(* CODESYS project lclsvacuum.library
   Company: SLAC
   Title: LCLSVacuumLib
   Description: No serial drivers exist in this library. Need LCLSVacuumSerialDrivers for that.
      1.2.0 ecat diagnostic
      1.2.1 added the ecat lib in here
      1.2.2 adding the ratio check function for valve interlocking
      1.3.6 added 275 & 500 gauges, minor changes
      1.4.0 added a normally open gate valve structure and FB
      1.5.0 added error and warning codes to ptm structure for pfeiffers
      1.5.1 seamless override open/close on vgc during transition from override to normal mode.
      1.7.0 ST_PTM now uses inheritence model.  Started implementing Ebara support.
      1.8.0 Moved to seperate functions for 937A and 937B controllers.
   Placeholder: LCLSVacuumLib
   Author: Alex Wallace & Scott Stubbs
   Version: 1.10.3

Project tree, tasks and I/O mapping:
  libraries: Tc2_EtherCAT, * (Beckhoff Automation GmbH); Tc2_Standard, * (Beckhoff Automation GmbH); Tc2_System, * (Beckhoff Automation GmbH); Tc2_TcpIp, * (Beckhoff Automation GmbH); Tc2_Utilities, * (Beckhoff Automation GmbH); Tc3_Interfaces, * (Beckhoff Automation GmbH); Tc3_Module, * (Beckhoff Automation GmbH)
  Data types/
    Gauges/
      data type E_PressureState
      data type Gauge_Type
      data type ST_VG
    Logger/
      data type E_MesgSevr
      data type E_MessengerState
      data type E_Subsystem
    Misc/
      data type ST_fbDiagnostics
      data type System_Struct
    Pumps/
      data type ST_AgilentControlStatus
      data type ST_EbaraDryPump
      data type ST_EbaraPTM
      data type ST_LeyboldPTM
      data type ST_PfeifferPTM
      data type ST_PTM
      data type ST_RoughPump
    Valves/
      data type E_VCN
      data type E_VGC
      data type ST_VCC
      data type ST_VCN
      data type ST_VGC
      data type ST_VGC_NO
      data type ST_VRC
    data type ISG_Struct
    data type ST_Encoder
    data type ST_LaserGate
    data type UpStrInVac_Struct
    data type UpStrOutVac_Struct
  Global Variables/
    global variables Constants
    global variables Global_Variables
    global variables GVL_Logger
  POUs/
    Functions/
      Gauge FB/
        function block FB_275 [ST]
        function block FB_500 [ST]
        function block FB_903 [ST]
        function block FB_907 [ST]
        function block FB_909 [ST]
        function block FB_925 [ST]
        function block FB_937A_VG [ST]
        function block FB_937B_VG [ST]
        function block FB_972 [ST]
        function block FB_Dumb_Gauge [ST]
        function block FB_GCM [ST]
        function block FB_GGO [ST]
        function block FB_GGO_dep [ST]
        function block FB_PressureState [ST]
      Pumps/
        function block FB_EbaraDryPump [ST]
        function block FB_PTM_Agilent [ST]
        function block FB_PTM_Ebara [ST]
        function block FB_PTM_LeyboldTD20Classic [ST]
        function block FB_PTM_MagDriveDigital [ST]
        function block FB_PTM_Pfeiffer [ST]
      Valve FB/
        function F_TURBO_VRC_ILK [ST]
        function F_VALVE_REL_ILK [ST]
        function F_VRC_DIODE_ILK [ST]
        function block FB_VCC [ST]
        function block FB_VCN [ST]
        function block FB_VGC [ST]: ACT_ResetAlarms
        function block FB_VGC_NO [ST]: ACT_ResetAlarms
        function block FB_VRC [ST]
        function block FB_VRC_OK_CLS [ST]
      function block FB_EcatDiag [ST]
      function block FB_Index [ST]: Dec, Inc, ValInc
    Logger/
      function block FB_Logger [ST]: Manager, SocketSendTo
      function block FB_LogMessage [ST]
      function SYSTEM_TIME_TO_RFC3339 [ST]
    program LOGGER [ST]
    program MAIN [ST]
  Version/
    global variables Global_Version
  Visualizations/
  00000000-0000-0000-0000-000000000000|LCLSVacuum.tmc
  LCLSVacuum.tmc
*)

// Data types/Gauges/E_PressureState
TYPE E_PressureState :
(
	Valid := gc_GaugeValidState,
	ValidHi	:= 1, //gc_GaugeValidState + 1,
	ValidLo	:= 2, //gc_GaugeValidState + 2,
	
	// Invalid states
	Invalid	:= -1, //gc_GaugeValidState - 1,
	Disconnected	:=	-2, //gc_GaugeValidState -2,
	OoR	:= -6, //gc_GaugeValidState -6,
	// Ion gauges
	Off		:= -3, //gc_GaugeValidState - 3,
	Starting	:= -4 //gc_GaugeValidState - 4
) INT;
END_TYPE

// Data types/Gauges/Gauge_Type
TYPE Gauge_Type: ( 
PG722B := 0, 
IG903 := 1 , 
PG907 := 2 , 
IG909:= 3 ,
PG925 := 4 );
(* This enumeration should match up with the EDM MUX button on the vacuum gauge expert controls screen *)
END_TYPE

// Data types/Gauges/ST_VG
TYPE ST_VG :
STRUCT
	/// A general gauge structure is used to make the rest of the interlocking simpler. There are some parameters for cold cathodes that are not used by pirani.
	///These features aren't disabled, they just aren't used, think child/parent classes. 
	/// Readbacks 
	rPRESS: REAL; //This is the human-readable pressure
	iPRESS_R: INT;
	xAT_VAC: BOOL;
	xPRESS_OK: BOOL;
	wState	:	WORD; //current gauge state, to be used as replacement for press OK bit in the future.
	(* 00 controller not on
		01 normal, aka pressure OK
		02 LO, pressure too low
		03 HI, pressure too high
		04 Gauge disconnected, HV off, no sensor detected, controller powering up
		05 cold cathode warming up
		*)
	eState	:	E_PressureState;
	
	/// Controls 
	xHV_DIS: BOOL;
	xHV_SW: BOOL;
	wHV_RO: WORD;
	
	/// Bakeout bit 
	xBAKEOUT: BOOL;
	
	eTYPE: Gauge_Type := PG907;
	iTYPE : INT := 0;
	wPG: WORD;
	
	/// Turn on Timers for cold cathode warmup 
	xTurnOnTime: BOOL;
	/// At vacuum setpoint for all gauges
	rVAC_SP: REAL := 0.5;
	/// Protection setpoint for ion gauges at which the gauge turns off, not used for pirani 
	rPRO_SP: REAL := 0.01;
	/// Protection setpoint hysteresis 
	rHYS_PR: REAL;
	/// Full scale pressure in Torr for baratron pressure conversion 
	rFULL_SCALE: REAL := 1000;
END_STRUCT
END_TYPE

// Data types/Logger/E_MesgSevr
TYPE E_MesgSevr :
(
	Emergency := 0, //system is unusable
	Alert	:= 1,	//action must be taken immediately
	Critical:= 2,	//critical conditions
	Error	:= 3,	//error conditions
	Warning	:= 4,	//warning conditions
	Notice	:= 5,	//normal but significant condition
	Info	:= 6,	//informational messages
	Debug	:= 7	//debug-level messages
) WORD;
END_TYPE

// Data types/Logger/E_MessengerState
TYPE E_MessengerState :
(
	Init := 0,
	CreateSocket	:= 1,
	Active	:= 2,
	CloseSocket := 3,
	Err	:= 10
);
END_TYPE

// Data types/Logger/E_Subsystem
TYPE E_Subsystem :
(
	NILVALUE := 0,
	VACUUM := 1,
	MPS := 2,
	MOTION := 3,
	FIELDBUS := 4,
	SDS := 5
)WORD;
END_TYPE

// Data types/Misc/ST_fbDiagnostics
TYPE ST_fbDiagnostics :
STRUCT
	asResults	:	ARRAY [1..20] OF STRING;
	resultIdx	:	FB_Index := (
		InitVal := 1,
		UpperLimit := 20
	);
	fString	:	FB_FormatString;
END_STRUCT
END_TYPE

// Data types/Misc/System_Struct
TYPE System_Struct :
STRUCT

	xswAlmRst 		: BOOL;(* Global Alarm Reset - EPICS Command *)
	xAtVacuum 	    : BOOL;(* System At Vacuum *)
	xFirstScan	    : BOOL; (* Bit set for one scan only during startup. Used for initialization. *)
	xOverrideMode	: BOOL; //This bit is set when using the override features of the system
	xIOState        : BOOL; (* ECat Bus Health *)

END_STRUCT
END_TYPE

// Data types/Pumps/ST_AgilentControlStatus
TYPE ST_AgilentControlStatus :
STRUCT

(* Inputs *)
	xdiR1   		:  BOOL;
	xdiLSpd 		:  BOOL;
	xdiStart		:  BOOL;
	xdiR2   		:  BOOL;
	xdiFlt   	:  BOOL;
	xswStart		:  BOOL;
	xswLSpd 		:  BOOL;
	xswSS   		:  BOOL;
	xilkStart	:  BOOL;
	xilkLSpd   	:  BOOL;
	xilkEnb   	:  BOOL;
	xilkSS   	:  BOOL;
	xAlmRst   	:  BOOL;

(* Outputs *)
	xdoStart	:  BOOL;
	xdoLSpd	:  BOOL;
	xdoEnb	:  BOOL;
	xdoSS	:  BOOL;

(* Alarm Outputs *)
	xalmFlt		:  BOOL;
	xalmStart	:  BOOL;
	xalmLSpd		:  BOOL;
	xalmSS		:  BOOL;
	xAlmSum		: BOOL;


END_STRUCT
END_TYPE

// Data types/Pumps/ST_EbaraDryPump
TYPE ST_EbaraDryPump EXTENDS ST_RoughPump :
STRUCT
(* Extension of the rough pump archetype for ebara 
Applicable to: 
EV-S20
EV-S50
EV-S100
EV-S200
*)

//Controls
q_xMPStart	:	BOOL; //Main Pump start
q_xBPStart	:	BOOL; // Booster Pump start (this can be started by the pump automatically)

xBPIlk	:	BOOL;	//Booster pump interlock
rBPIlkSP	:	REAL := 30; //Booster pump pressure setpoint
tonBP	:	TON := (PT:=T#5S); //Timer for pressure and valve stability


//Readbacks
i_xMPStatus	:	BOOL; //MP status
i_xBPStatus	:	BOOL; //BP status
i_xWarning	:	BOOL; //Warning status
i_xAlarm	:	BOOL; //Alarm, maps to error
i_xRemote	:	BOOL; //Remote control status


END_STRUCT
END_TYPE

// Data types/Pumps/ST_EbaraPTM
TYPE ST_EbaraPTM EXTENDS ST_PTM :
STRUCT
(* Extension of the PTM archetype for Ebara turbo controllers 
Applicable to: 
ETC series
*)
//Controls
i_xStart   : BOOL; //Momentary start switch
i_xStop    : BOOL; //Momentary stop switch
//i_xReset   : BOOL; //Momentary reset switch - resets protection functions
q_xStart   : BOOL; //Outputs - FB decides if these are actually set
q_xStop    : BOOL;
q_xReset   : BOOL;
q_xProtection : BOOL; //NC. If opened, pump will decelerate/not start

iq_xSpeedSet    : BOOL; //Request to set speed
q_iSpeedSet   : DINT; //Requested speed (min. 100 RPM)

i_xOverride   : BOOL; //Override mode - ignores interlocks

//Readbacks - also has Accel/At speed/Decel/Fault/Cur Speed (min 100RPM)
i_xRotate : BOOL; //If open, pump is rotating
i_xDecel  : BOOL; //If closed, brake engaged (pump decelerating)
i_xNCFault  : BOOL; //Normally closed fault wiring. If false, there is a fault, or cable is unplugged.
i_iRawSpeed	:	INT; //Raw pump speed from analog input

END_STRUCT
END_TYPE

// Data types/Pumps/ST_LeyboldPTM
TYPE ST_LeyboldPTM EXTENDS ST_PTM :
STRUCT
(* Extension of the PTM archetype for Oerlikon turbo controllers 
Applicable to: 
Mag Drive Digital
Mag Drive S
More?
*)
//Readbacks
	i_xDecel	:	BOOL;
	i_diPumpTemp:	DINT;
	i_diPwr   	:   DINT;
	i_diElecTemp:	DINT;
	i_xTempFault:	BOOL;
	i_xNCError	:	BOOL; //Using normally closed wiring

//Controls
	q_xRemote : BOOL; (* Remote control enabled *)
END_STRUCT
END_TYPE

// Data types/Pumps/ST_PfeifferPTM
TYPE ST_PfeifferPTM EXTENDS ST_PTM :
STRUCT
(* Extension of the PTM archetype for Pfeiffer turbos 
Applicable to: 
HiPace series w/ onboard controllers
More?
*)
//Readbacks
	i_diPwr		:	DINT;
	i_diElecTemp	:	DINT;
	i_diBtmTemp:	DINT;
	i_diBrngTemp:	DINT;
	i_diMtrTemp:	DINT;
	i_iErrorCode	:	INT; //might change these to enumeration someday
	i_iWarningCode	:	INT;
	i_xTempFault	:	BOOL;
	
END_STRUCT
END_TYPE

// Data types/Pumps/ST_PTM
TYPE ST_PTM :
STRUCT
(* General PTM Structure
Each PTM might have a serial control structure, but all will have a general supervisory control structure

NOTE: This is an archetype, use an extension of this structure for a specific pump (or make one).

*)

(* Controls *)
	i_xRunSW	:	BOOL;
	i_xReset	:	BOOL; //For resetting faults
	q_RunDO 	:	BOOL;

(* Readbacks *)
	xExtRunOk	:	BOOL; (* also a control *)
	i_xAccel	:	BOOL;
	i_xAtSpd	:	BOOL;
	i_iCurSpd	:	DINT;
	
	xCommTimeout	:	BOOL := TRUE;  (* Initialized true since we haven't talked to pump yet *)
(* Alarm Outputs *)
	xFault		:	BOOL; //Note, for Ebara this is *false* in a fault condition!
	xWarn		:	BOOL; (* warning *)
	
(* IWS instructions *)
	xActive	:	BOOL; // this bit is set to add the pump to the system
	iPumpGrp 	:	INT; // all members of a pump group start at the same time

END_STRUCT
END_TYPE

// Data types/Pumps/ST_RoughPump
TYPE ST_RoughPump :
STRUCT
	
(* Generic roughing pump controls 

NOTE: This is an archetype, use an extension of this structure for a specific pump (or make one).

*)

//Controls
i_xRunSW	:	BOOL; //epics/ software control switch

//Status and Readback
xIlk	:	BOOL; //Interlock bit, true means OK to run
xExtIlk	:	BOOL; //External interlock, this is where the logic goes
xAtSpd	:	BOOL; //Pump at speed setpoint

xWrn	:	BOOL; //Pump warning
iWrn	:	BOOL; //Warning state/code
xErr	:	BOOL; //Error summary
iErr	:	BOOL; //Error state/code

END_STRUCT
END_TYPE

// Data types/Valves/E_VCN
TYPE E_VCN :
	(
CloseValve	:= 0,
ControlValve	:= 1,
OpenValve	:= 2
	);
END_TYPE

// Data types/Valves/E_VGC
TYPE E_VGC :
(

	Vented,
	AtVacuum,
	ERR_DiffPress,
	ERR_LostVac

);
END_TYPE

// Data types/Valves/ST_VCC
TYPE ST_VCC :
STRUCT

(* Inputs *)
	xOPN_SW	: BOOL;
	xOvrdOpn	:	BOOL;
	xOPN_OK	: BOOL;

(* Outputs *)
	xOPN_DO	: BOOL;

END_STRUCT
END_TYPE

// Data types/Valves/ST_VCN
TYPE ST_VCN :
STRUCT
	(* VCN - Valve Controlled Needle
	Used for Pfeiffer EVR 116 needle valves *)
	// Inputs
	i_iPosition	:	INT; //Position readback (if it exists)
	
	// Outputs
	q_iRawPosition	:	INT; //Position control 
	//For the EVR 116 this is 0-10V analog
	
	//Softvariables
	xIlk	:	BOOL := FALSE; // Interlock Bit
	rUpperLimit	:	REAL;	//Upper limit on valve open
	rReqPosition	:	REAL; //Requested position (0.0-100.0%)
	eValveControl	:	E_VCN := CloseValve; // Valve control state

	ftIlk	:	F_TRIG;	

END_STRUCT
END_TYPE

// Data types/Valves/ST_VGC
TYPE ST_VGC :
STRUCT

(* Readbacks *)
	i_xOpnLS	: BOOL;
	i_xClsLS	: BOOL;

(* EPICS Controls *)
	xOPN_SW	: BOOL;
	xAlmRst	: BOOL;
	xOvrdOpn	:	BOOL;

(* Interlocks *)
	xDP_OK	:	BOOL;	// Indicates the valve can be opened because the differential pressure is low enough
	xEXT_OK	:	BOOL := FALSE;	(* External interlock for custom interlocking in addition to regular DP ilk, this must be set true, or the interlock condition before calling the FB_VGC *)
	xOPN_OK	:	BOOL;	(* Final SUM of DP_OK and EXT_OK, needed because it allows the DP ilk to be switched off, see FB_VGC.Dis_DPIlk *)
	
rAT_VAC_SP	:	REAL;	// Interlock setpoint for gauges on both sides of valve
	rAT_VAC_SP_LAST	:	REAL;	// Interlock setpoint for gauges on both sides of valve
	rAT_VAC_HYS	:	REAL;	// Hysteresis of the vacuum sp
	rHYST_PERC	:	REAL;	// Hysteresis percentage
	xAT_VAC	:	BOOL;	//At vacuum setpoint

(* Controls *)
	xOPN_DO	: BOOL;

(* Alarm Outpus *)
	xERR_DifPres		: 	BOOL;
	xERR_LstVac		: 	BOOL;
	xAlmSum			: 	BOOL;

END_STRUCT
END_TYPE

// Data types/Valves/ST_VGC_NO
TYPE ST_VGC_NO EXTENDS ST_VGC :
STRUCT
	(* A normally open gate valve needs permission to close! *)
	(* EPICS Controls *)
	xCLS_SW	:	BOOL;
	xOvrdCls	:	BOOL;
	
	(* Interlocks *)
	xCLS_OK	:	BOOL;
	
	(* IO Controls *)
	xCLS_DO	:	BOOL;
	
	
END_STRUCT
END_TYPE

// Data types/Valves/ST_VRC
TYPE ST_VRC :
STRUCT
(* Readbacks *)
	i_xOpnLS	:	BOOL;
	i_xClsLS	:	BOOL;

(* Inputs *)
	xOPN_SW	: BOOL;
	xOvrdOpn	:	BOOL;
	xOPN_OK	: BOOL;
	xCLS_OK : BOOL := TRUE;
(* Outputs *)
	xOPN_DO	: BOOL;

END_STRUCT
END_TYPE

// Data types/ISG_Struct
TYPE ISG_Struct :
STRUCT

	xdoHV1 : BOOL;
	xdoHV2 : BOOL;
	xdoHV3 : BOOL;

	xswHV1 : BOOL;
	xswHV2 : BOOL;
	xswHV3 : BOOL;

	xilkHV1 : BOOL;
	xilkHV2 : BOOL;
	xilkHV3 : BOOL;

END_STRUCT
END_TYPE

// Data types/ST_Encoder
TYPE ST_Encoder :
STRUCT
	xENC_PWR_SW : BOOL;
	xENC_PWR : BOOL;
END_STRUCT
END_TYPE

// Data types/ST_LaserGate
TYPE ST_LaserGate :
STRUCT
	xIN	:	BOOL;
END_STRUCT
END_TYPE

// Data types/UpStrInVac_Struct
TYPE UpStrInVac_Struct :
STRUCT

	xdiUpSVac : BOOL;

END_STRUCT
END_TYPE

// Data types/UpStrOutVac_Struct
TYPE UpStrOutVac_Struct :
STRUCT

	xdoUpSVac : BOOL;
	xilkUpSVac : BOOL;

END_STRUCT
END_TYPE

// Global Variables/Constants
VAR_GLOBAL CONSTANT
	gc_iSizeOfGGOArray : INT := 50;
	gc_GaugeValidState :	INT := 0;
END_VAR

// Global Variables/Global_Variables
VAR_GLOBAL
	g_iSizeOfGGOArray : INT := 50;
	
	g_stSystem	:	System_Struct;
	
	g_DummyVG	:	ST_VG;
	
END_VAR

// Global Variables/GVL_Logger
VAR_GLOBAL
	g_psLogHost	: T_IPv4Addr := '172.21.32.9';
	g_udpSyslog	:	UDINT := 514;
	gMesgBuffer	:	ARRAY [0..cMesgArraySize] OF T_MaxString; //maybe this should be persistent...
	gsCurrentTime	:	T_MaxString := cNILVALUE;
	gsHostName	:	T_MaxString := cNILVALUE;
	fbLogMessage : FB_LogMessage;
	gfbBuffer 			:	FB_StringRingBuffer;
END_VAR
VAR_GLOBAL CONSTANT
	acsSubsystems	:	ARRAY [0..5] OF STRING := 
	['-', 'VACUUM', 'MPS', 'MOTION', 'FIELDBUS', 'SDS'];
	cNILVALUE	:	STRING(1) := '-';
	cMesgArraySize : INT := 50;
	cwFacility: WORD := 20; // local4
	// Syslog Version
	cwSyslogVer: WORD := 1;
END_VAR

// Version/Global_Version
{attribute 'TcGenerated'}
// This function has been automatically generated from the project information.
VAR_GLOBAL CONSTANT
	{attribute 'const_non_replaced'}
	{attribute 'linkalways'}
	stLibVersion_LCLSVacuumLib : ST_LibVersion := (iMajor := 1, iMinor := 10, iBuild := 3, iRevision := 0, sVersion := '1.10.3');
END_VAR

// POUs/Functions/Gauge FB/FB_275
FUNCTION_BLOCK FB_275
VAR_IN_OUT
	PG : ST_VG;
END_VAR
VAR_INPUT
END_VAR
VAR_OUTPUT
END_VAR
VAR

	MinPressure: REAL := 1E-4;

	V : REAL;

END_VAR

(* This function block is used to provide protection and automatic turn on of ion gauges,
 it also manages the turn on of the AT_VAC boolean, and checks to make sure the pressure is good *)
(* For MKS 275 mini-convectron *)


(* Real-value calculation *)

V := 10*INT_TO_REAL(PG.iPRESS_R)/32767;	

IF V > 0.36 AND V < 0.38 THEN

PG.rPRESS := MinPressure;

ELSIF V >= 0.38 AND V < 2.842 THEN

PG.rPRESS := LREAL_TO_REAL( -0.02585 + 0.03767*V + 0.04563*EXPT(V,2)+ 0.1151*EXPT(V,3) - 0.04158*EXPT(V,4)+ 0.008737*EXPT(V,5));

ELSIF V >= 2.842 AND V < 4.945 THEN

PG.rPRESS := LREAL_TO_REAL((0.1031-0.02322*V+0.07229*EXPT(V,2))/(1-0.3986*V+0.07438*EXPT(V,2)-0.006866*EXPT(V,3)));

ELSIF V >= 4.945 THEN

PG.rPRESS := LREAL_TO_REAL((100.624-20.5623*V)/(1-0.37679*V+0.0348656*EXPT(V,2)));

END_IF

(* Protection Functions *)
(* If the PG pressure is greater than the IG.PRO_SP then the gauge is disabled *)
(* If the PG pressure is less than the IG.PRO_SP then the gauge is enabled *)
(* This FB also implements some hysteresis so the gauge doesn't have rapid power cycling while near the turn on boundary *)

(* Pressure OK check *)
PG.xPRESS_OK := (PG.rPRESS >= MinPressure);

(* Setpoint evaluation *)
PG.xAT_VAC := PG.xPRESS_OK AND (PG.rPRESS<PG.rVAC_SP);

END_FUNCTION_BLOCK

// POUs/Functions/Gauge FB/FB_500
FUNCTION_BLOCK FB_500
VAR_IN_OUT
	IG : ST_VG;
END_VAR
VAR_INPUT
	PG	:	ST_VG;
END_VAR
VAR_OUTPUT
	xHV_SW: BOOL;
	rPRESS: INT;
	rVAC_SP: INT;
END_VAR
VAR
	rV : REAL;
	GaugeTurnOnTmr : TON;
	MinPressure: REAL := 1E-9;
	
END_VAR
VAR CONSTANT
	cDefaultPressure : REAL := 750.0;
	vBase	:	REAL := 1; //corresponding vbase 1V actually?
	pBase	:	REAL := 1.0E-9; //i think the pbase might be 1E-9 for the default curve...
	vSlope	:	REAL := 1.0; //looks correct for default curve
END_VAR

(* 500 Logarithmic Output Conversion, factory default configuration *)

rV := 10*INT_TO_REAL(IG.iPRESS_R)/32767;

IF rV >= 0.5 AND rV < 1.0  THEN
	IG.wState := 5;
	IG.eState := Starting;
	IG.rPRESS := cDefaultPressure;
ELSIF rV < 0.4 THEN
	IG.wState := 4;//HV Off/ gauge disconnected
	IG.eState := Off;
	IG.rPRESS := cDefaultPressure;
ELSE
	IG.wState := 1;
	IG.eState := Valid;
	IG.rPRESS := LREAL_TO_REAL(EXPT(10,((rV-vBase)/vSlope+LOG(pBase))));
END_IF



(* Ion Gauge Protection Functions *)
(* If the PG pressure is greater than the VG.PRO_SP then the gauge is disabled *)
(* If the PG pressure is less than the VG.PRO_SP then the gauge is enabled *)
(* This FB also implements some hysteresis so the gauge doesn't have rapid power cycling while near the turn on boundary *)

IF PG.rPRESS < IG.rPRO_SP AND PG.xPRESS_OK THEN

	IG.xHV_DIS := IG.xHV_SW;

ELSIF IG.xHV_DIS THEN
	IF IG.rPRESS > (IG.rPRO_SP + IG.rHYS_PR)  OR PG.rPRESS > (IG.rPRO_SP + IG.rHYS_PR) THEN
		IG.xHV_DIS := FALSE;
		IG.xHV_SW := FALSE;
	END_IF
ELSE
	IG.xHV_DIS := FALSE;
	IG.xHV_SW := FALSE;
END_IF

(* Pressure gauge OK checks *)

//Backwards compatibility
IG.xPRESS_OK := (IG.wState = 1) OR IG.xBAKEOUT;

(* Setpoint evaluation *)
IG.xAT_VAC := (IG.xPRESS_OK AND (IG.rPRESS < IG.rVAC_SP)) OR IG.xBAKEOUT;

END_FUNCTION_BLOCK

// POUs/Functions/Gauge FB/FB_903
FUNCTION_BLOCK FB_903
VAR_IN_OUT

	IG : ST_VG;

END_VAR
VAR_INPUT

	PG : ST_VG;

END_VAR
VAR_OUTPUT
END_VAR
VAR
	rMaxPressure: REAL := 5E-3;
	rMinPressure: REAL := 3E-10;

	V: REAL;

	GaugeTurnOnTmr : TON;
	fbGaugeState : FB_PressureState;
END_VAR

(* This function block is used to provide protection and automatic turn on of ion gauges,
 it also manages the turn on of the AT_VAC boolean, and checks to make sure the pressure is good *)

(* Real-value calculation *)
(* Generic expression for pressure in the MKS systems

P = 10^(V/0.6 -12)

*)

V := 10*INT_TO_REAL(IG.iPRESS_R)/32767;

IG.rPRESS := LREAL_TO_REAL(EXPT(10,(V-11)));


(* Protection Functions *)
(* If the PG pressure is greater than the IG.PRO_SP then the gauge is disabled *)
(* If the PG pressure is less than the IG.PRO_SP then the gauge is enabled *)
(* This FB also implements some hysteresis so the gauge doesn't have rapid power cycling while near the turn on boundary *)

IF PG.rPRESS < IG.rPRO_SP AND PG.xPRESS_OK THEN

	IG.xHV_DIS := IG.xHV_SW;

ELSIF IG.xHV_DIS THEN
	IF (IG.rPRESS > (IG.rPRO_SP + IG.rHYS_PR)) OR PG.rPRESS > (IG.rPRO_SP + IG.rHYS_PR) THEN
		IG.xHV_DIS := FALSE;
		IG.xHV_SW := FALSE;
	END_IF
ELSE
	IG.xHV_DIS := FALSE;
	IG.xHV_SW := FALSE;
END_IF

(* Pressure OK check *)
fbGaugeState.i_rV := V;
fbGaugeState.i_MaxPressure := rMaxPressure;
fbGaugeState.i_MinPressure := rMinPressure;
fbGaugeState(iq_stVG:=IG);

(* Setpoint evaluation *)
IG.xAT_VAC := (IG.xPRESS_OK AND (IG.rPRESS<IG.rVAC_SP)) OR IG.xBAKEOUT;

END_FUNCTION_BLOCK

// POUs/Functions/Gauge FB/FB_PressureState
FUNCTION_BLOCK FB_PressureState
VAR_INPUT
	i_rV	:	REAL;
	i_rVMin	:	REAL := 0.01; // Anything less than this voltage is considered disconnected
	i_rVMax :	REAL := 10.5; // Anything more than this is considered invalid
	i_IGTurnOnTime	:	TIME := T#10S;
	
	i_MinPressure	:	REAL;
	i_MaxPressure	:	REAL;
END_VAR
VAR_OUTPUT
	q_eState 	:	E_PressureState;
END_VAR
VAR_IN_OUT
	iq_stVG	:	ST_VG;
END_VAR
VAR
	tonGaugeTurnOnTmr : TON;
END_VAR

(* Pressure State Evaluation
A. Wallace, 2016-8-31

This FB serves to evaluate the state of the pressure based on the raw voltage, pressure, and gauge state.

*)
// Is the gauge plugged in, and within a reasonable range?
IF i_rV < i_rVMin THEN
	q_eState := Disconnected;
ELSIF i_rV > i_rVMax THEN
	q_eState := Invalid;
ELSE
	// Is the gauge reading back a pressure that makes sense?
	CASE iq_stVG.eTYPE OF
		IG903:
			tonGaugeTurnOnTmr(IN:=iq_stVG.xHV_DIS, PT:=i_IGTurnOnTime, Q=>iq_stVG.xTurnOnTime);
			IF iq_stVG.xHV_DIS THEN
				IF tonGaugeTurnOnTmr.Q THEN
					IF iq_stVG.rPRESS >= i_MinPressure AND iq_stVG.rPRESS <= i_MaxPressure THEN
						q_eState := Valid;
					ELSE
						q_eState := OoR; 
					END_IF
				ELSE
						q_eState := Starting;
				END_IF
			ELSE
				q_eState := Off;
			END_IF
		IG909:
			IF iq_stVG.xHV_DIS THEN
				IF iq_stVG.rPRESS >= i_MinPressure AND iq_stVG.rPRESS <= i_MaxPressure THEN
					q_eState := Valid;
				ELSE
					q_eState := OoR;
				END_IF
			ELSE
				q_eState := Off;
			END_IF
		PG907, PG925, PG722B:
			IF iq_stVG.rPRESS >= i_MinPressure AND iq_stVG.rPRESS <= i_MaxPressure THEN
				q_eState := Valid;
			ELSIF iq_stVG.rPRESS < i_MinPressure THEN
				q_eState := ValidLo;
			ELSE
				q_eState := ValidHi;
			END_IF
		ELSE
			q_eState := Invalid;
	END_CASE
END_IF


iq_stVG.eState := q_eState;

// Legacy Press OK boolean eval
iq_stVG.xPRESS_OK := q_eState >= gc_GaugeValidState;

END_FUNCTION_BLOCK

// POUs/Functions/Gauge FB/FB_907
FUNCTION_BLOCK FB_907
VAR_IN_OUT

	PG : ST_VG;

END_VAR
VAR_INPUT
END_VAR
VAR_OUTPUT
END_VAR
VAR
	V : REAL;
	A : REAL := 3.29;
	B : REAL := 24.98;
	C : REAL  := 0.98;
	V_0 : REAL := 0.3752;
	D: REAL := 4.929;
	F: REAL := 1.6E-6;
	G: REAL := -225;
	H: REAL := 2.0253;
	K: REAL := 0.52703;
	
	fbGaugeState : FB_PressureState;
	// Torr
	rMaxPressure: REAL := 1000;
	// Torr
	rMinPressure: REAL := 1E-3;
END_VAR

(* This function block is used to provide protection and automatic turn on of ion gauges,
 it also manages the turn on of the AT_VAC boolean, and checks to make sure the pressure is good *)


(* Real-value calculation *)

V := 10*INT_TO_REAL(PG.iPRESS_R)/32767;

IF V > 0.38 AND V < 4.85 THEN

PG.rPRESS := LREAL_TO_REAL(EXPT((A/(B/(EXPT(V,2)-EXPT(V_0,2)-1))), 1/C));

ELSIF V > 4.85 AND V < 5.18 THEN

PG.rPRESS := LREAL_TO_REAL(SQRT( ( (V-D)+SQRT(EXPT((V-D),2)-4*F*G ))/(2*F) ));

ELSIF V> 5.18 THEN

PG.rPRESS := EXP((V-H)/K);

END_IF

(* Pressure OK check *)
fbGaugeState.i_rV := V;
fbGaugeState.i_MaxPressure := rMaxPressure;
fbGaugeState.i_MinPressure := rMinPressure;
fbGaugeState(iq_stVG:=PG);


(* Setpoint evaluation *)
PG.xAT_VAC := PG.xPRESS_OK AND (PG.rPRESS<PG.rVAC_SP) OR PG.xBAKEOUT;

END_FUNCTION_BLOCK

// POUs/Functions/Gauge FB/FB_909
FUNCTION_BLOCK FB_909
VAR_IN_OUT

	IG : ST_VG;

END_VAR
VAR_INPUT

	PG : ST_VG;

END_VAR
VAR_OUTPUT
END_VAR
VAR
	rMaxPressure: REAL := 5E-2;
	rMinPressure: REAL := 3E-10;

	V: REAL;
	fbGaugeState : FB_PressureState;
END_VAR

(* This function block is used to provide protection and automatic turn on of ion gauges,
 it also manages the turn on of the AT_VAC boolean, and checks to make sure the pressure is good *)

(* Real-value calculation *)
(* Generic expression for pressure in the MKS systems

P = 10^(V/0.6 -12)

*)

V := 10*INT_TO_REAL(IG.iPRESS_R)/32767;

IG.rPRESS := LREAL_TO_REAL(EXPT(10,(V-10)));


(* Protection Functions *)
(* If the PG pressure is greater than the IG.PRO_SP then the gauge is disabled *)
(* If the PG pressure is less than the IG.PRO_SP then the gauge is enabled *)
(* This FB also implements some hysteresis so the gauge doesn't have rapid power cycling while near the turn on boundary *)

IF PG.rPRESS < IG.rPRO_SP AND PG.xPRESS_OK THEN

	IG.xHV_DIS := IG.xHV_SW;

ELSIF IG.xHV_DIS THEN
	IF IG.rPRESS > IG.rPRO_SP + IG.rHYS_PR OR PG.rPRESS > IG.rPRO_SP + IG.rHYS_PR THEN
		IG.xHV_DIS := FALSE;
		IG.xHV_SW := FALSE;
	END_IF
ELSE
	IG.xHV_DIS := FALSE;
	IG.xHV_SW := FALSE;
END_IF

(* Pressure OK check *)
fbGaugeState.i_rV := V;
fbGaugeState.i_MaxPressure := rMaxPressure;
fbGaugeState.i_MinPressure := rMinPressure;
fbGaugeState(iq_stVG:=IG);

(* Setpoint evaluation *)
IG.xAT_VAC := (IG.xPRESS_OK AND (IG.rPRESS<IG.rVAC_SP)) OR IG.xBAKEOUT;

END_FUNCTION_BLOCK

// POUs/Functions/Gauge FB/FB_925
FUNCTION_BLOCK FB_925
VAR_INPUT
END_VAR
VAR_OUTPUT
END_VAR
VAR_IN_OUT
	VG	: ST_VG;
END_VAR
VAR
	rV : REAL;
	fbGaugeState : FB_PressureState;
	rMaxPressure	:	REAL := 760; //Torr
	rMinPressure	:	REAL := 1E-5; //Torr
END_VAR

(* Standard MKS 9XX series conversion *)
(* works for 972 and 925 *)

rV := 10*INT_TO_REAL(VG.iPRESS_R)/32767;

IF rV >= 1 THEN
	VG.rPRESS := LREAL_TO_REAL(EXPT(10, rV-6));
	VG.xPRESS_OK := TRUE;
	VG.wState := 1;
ELSIF rV >= 0.99 AND rV < 1 THEN
	VG.rPRESS := 1E-5;
	VG.xPRESS_OK := TRUE;
	VG.wState := 1;
ELSE
	VG.xPRESS_OK := FALSE;
	VG.wState := 2;
END_IF

(* Pressure OK check *)
fbGaugeState.i_rV := rV;
fbGaugeState.i_MaxPressure := rMaxPressure;
fbGaugeState.i_MinPressure := rMinPressure;
fbGaugeState(iq_stVG:=VG);

(* Setpoint evaluation *)
VG.xAT_VAC := VG.xPRESS_OK AND (VG.rPRESS < VG.rVAC_SP);

END_FUNCTION_BLOCK

// POUs/Functions/Gauge FB/FB_937A_VG
FUNCTION_BLOCK FB_937A_VG
VAR_IN_OUT
	VG : ST_VG;
END_VAR
VAR_INPUT
	PG	:	ST_VG := g_DummyVG;
END_VAR
VAR_OUTPUT
END_VAR
VAR
	rV	:	REAL;
END_VAR

(* 937A Logarithmic Output Conversion *)
(* 7-15-2015 *)
(* This function will read the pressure from any gauge on a 937A. *)

rV := 10*INT_TO_REAL(VG.iPRESS_R)/32767;
VG.rPRESS := LREAL_TO_REAL(EXPT(10,rV/0.6-12));


(* Ion Gauge Protection Functions *)
(* If the PG pressure is greater than the VG.PRO_SP then the gauge is disabled *)
(* If the PG pressure is less than the VG.PRO_SP then the gauge is enabled *)
(* This FB also implements some hysteresis so the gauge doesn't have rapid power cycling while near the turn on boundary *)

IF PG.rPRESS < VG.rPRO_SP AND PG.wPG = 1 THEN

VG.xHV_DIS := NOT VG.xHV_SW;

ELSIF NOT VG.xHV_DIS THEN
	IF VG.rPRESS > VG.rPRO_SP + VG.rHYS_PR OR PG.rPRESS > VG.rPRO_SP + VG.rHYS_PR THEN
		VG.xHV_DIS := TRUE;
	END_IF
ELSE
	VG.xHV_DIS := TRUE;
END_IF


(* Pressure gauge OK checks *)
VG.xPRESS_OK := (rV <=9.6 ) AND (rV>=0.6); //legacy

IF (rV <=9.6 ) AND (rV>=0.6) THEN
	VG.wState := 1; // normal
ELSIF rV >= 0.18 AND rV <= 0.22 THEN
	VG.wState := 2; //LO
ELSIF rV >= 9.7 AND rV<= 9.9 THEN
	VG.wState := 3; //HIGH
ELSIF rV > 9.9 THEN
	VG.wState := 4; //other fault
ELSIF rV < 0.18 THEN
	VG.wState := 0; //not on
ELSE
	VG.wState := 9; // unknown state, something is really messed up
END_IF

(* Setpoint evaluation *)
VG.xAT_VAC := (VG.wState =1) AND VG.rPRESS < VG.rVAC_SP;

END_FUNCTION_BLOCK

// POUs/Functions/Gauge FB/FB_937B_VG
FUNCTION_BLOCK FB_937B_VG
VAR_IN_OUT
	VG : ST_VG;
END_VAR
VAR_INPUT
	PG	:	ST_VG := g_DummyVG;
END_VAR
VAR_OUTPUT
END_VAR
VAR
	rV	:	REAL;
END_VAR

(* 937B Logarithmic Output Conversion *)
(* 5-20-2016, Alex Wallace and Scott Stubbs *)
(* This function will read the pressure from any gauge on a 937B. *)

rV := 10*INT_TO_REAL(VG.iPRESS_R)/32767;
VG.rPRESS := LREAL_TO_REAL(EXPT(10,(rV-7.2)/0.6));


(* Ion Gauge Protection Functions *)
(* If the PG pressure is greater than the VG.PRO_SP then the gauge is disabled *)
(* If the PG pressure is less than the VG.PRO_SP then the gauge is enabled *)
(* This FB also implements some hysteresis so the gauge doesn't have rapid power cycling while near the turn on boundary *)

IF PG.rPRESS < VG.rPRO_SP AND PG.wPG = 1 THEN

VG.xHV_DIS := NOT VG.xHV_SW;

ELSIF NOT VG.xHV_DIS THEN
	IF VG.rPRESS > VG.rPRO_SP + VG.rHYS_PR OR PG.rPRESS > VG.rPRO_SP + VG.rHYS_PR THEN
		VG.xHV_DIS := TRUE;
	END_IF
ELSE
	VG.xHV_DIS := TRUE;
END_IF


(* Pressure gauge OK checks *)
VG.xPRESS_OK := (rV <=9.6 ) AND (rV>=0.6);

IF (rV <=9.7 ) AND (rV>=0.3) THEN
	VG.wState := 1; // normal
ELSIF rV >= 0.18 AND rV <= 0.22 THEN
	VG.wState := 2; //LO
ELSIF rV > 9.7 AND rV<= 9.9 THEN
	VG.wState := 3; //HIGH
ELSIF rV > 9.9 THEN
	VG.wState := 4; //other fault
ELSIF rV < 0.18 THEN
	VG.wState := 0; //not on
ELSE
	VG.wState := 9; // unknown state, something is really messed up
END_IF

(* Setpoint evaluation *)
VG.xAT_VAC := (VG.wState =1) AND VG.rPRESS < VG.rVAC_SP;

END_FUNCTION_BLOCK

// POUs/Functions/Gauge FB/FB_972
FUNCTION_BLOCK FB_972
VAR_INPUT
END_VAR
VAR_OUTPUT
END_VAR
VAR_IN_OUT
	VG	: ST_VG;
END_VAR
VAR
	rV : REAL;
END_VAR

(* Standard MKS 9XX series conversion *)
(* works for 972 and 925 *)

rV := 10*INT_TO_REAL(VG.iPRESS_R)/32767;

IF rV > 1 THEN
	VG.rPRESS := LREAL_TO_REAL(EXPT(10, 2*rV-11));
	VG.xPRESS_OK := TRUE;
	VG.wState := 1;
ELSE
	VG.xPRESS_OK := FALSE;
	VG.wState := 2;
END_IF

END_FUNCTION_BLOCK

// POUs/Functions/Gauge FB/FB_Dumb_Gauge
FUNCTION_BLOCK FB_Dumb_Gauge
VAR_IN_OUT
	iq_stPG : ST_VG;
END_VAR
VAR_INPUT
	i_stPGA : ST_VG;
	i_stPGB : ST_VG;
	i_stVRCA : ST_VRC;
	i_stVRCB : ST_VRC;
END_VAR
VAR_OUTPUT
END_VAR
VAR
END_VAR

(*
Alex Wallace 2013-10-28

The dummy gauge functions like so:
If my A side valve is open, I mimic the A side gauge.
If my B 	"	 			"			B	"		.
Else, I am at atmosphere, and my pressure is OK. 

The point of this gauge is to provide pressure readbacks for sections of the line that do not have gauges, and may move into an unknown pressure state.
*)

IF i_stVRCA.xOPN_DO THEN
iq_stPG := i_stPGA;
ELSIF i_stVRCB.xOPN_DO THEN
iq_stPG := i_stPGB;
ELSE
iq_stPG.xAT_VAC := FALSE;
iq_stPG.rPRESS := 750;
iq_stPG.xPRESS_OK := TRUE;
END_IF

END_FUNCTION_BLOCK

// POUs/Functions/Gauge FB/FB_GCM
FUNCTION_BLOCK FB_GCM
VAR_IN_OUT
	stVG	:	ST_VG;
END_VAR
VAR_OUTPUT
END_VAR
VAR
	rMinPressure: REAL;
	rV	:REAL;
END_VAR

(* Baratron Pressure Calc 
A. Wallace
2016-6-16
The full-scale pressure times the ratio of the meas.
voltage to full-scale voltage (10V).
The minimum pressure is always going to be 5e-4 * F.S.V.*)

rMinPressure := stVG.rFULL_SCALE * 5E-4;


rV :=MAX((10*INT_TO_REAL(stVG.iPRESS_R)/32767),0);
stVG.rPRESS := (stVG.rFULL_SCALE/10)*rV;
IF stVG.rPRESS > rMinPressure THEN
	stVG.xPRESS_OK := TRUE;
ELSE
	stVG.xPRESS_OK := FALSE;
END_IF

END_FUNCTION_BLOCK

// POUs/Functions/Gauge FB/FB_GGO
FUNCTION_BLOCK FB_GGO
VAR_IN_OUT
	iq_astGauges: ARRAY[0..gc_iSizeOfGGOArray] OF ST_VG;
	iq_axHV_RO: ARRAY[0..gc_iSizeOfGGOArray] OF BOOL;
END_VAR
VAR_INPUT
	i_iIndex: INT;
END_VAR
VAR

	stPG: ST_VG;
	stVG	:	ST_VG;

	
	// FBs
	fb903	:	FB_903;
	fb907	:	FB_907;
	fb909	:	FB_909;
	fb925	:	FB_925;
	fbGCM	:	FB_GCM;
	
END_VAR

(* This function block is used to calculate the pressure from the analog input voltage and to provide protection and automatic turn on of ion gauges.
 It also manages the turn on fo the AT_VAC boolean, and checks to make sure the pressure is good *)

(* Full-scale pressure conversion factor *)

(* Real-value voltage calculation *)
(* Generic expression for pressure in the MKS systems

P = 10^(V/0.6-12)

722B = 0
903 = 1
907 = 2
909 = 3
925 = 4

*)

stVG := iq_astGauges[LIMIT(0 ,i_iIndex, gc_iSizeOfGGOArray)];

IF WORD_TO_INT(stVG.wPG) <= gc_iSizeOfGGOArray THEN
	(* Check pressure gauge type before assignment *)
	(* Add high pressure gauge types here *)
		IF iq_astGauges[stVG.wPG].eTYPE = PG722B OR //722B
		iq_astGauges[stVG.wPG].eTYPE = PG907 OR //907
		iq_astGauges[stVG.wPG].eTYPE = PG925 THEN //925
			stPG := iq_astGauges[stVG.wPG];
			
		ELSE
			//Default to allow the IG to turn on, this allows someone to set the PG to another IG and turn the gauge on whenever they want
			stPG.rPRESS := 1E-3;
			stPG.xPRESS_OK := TRUE;
		END_IF
	
END_IF

CASE iq_astGauges[i_iIndex].eTYPE OF
	PG722B:
		fbGCM(stVG:=stVG);
	IG903:
		fb903(IG:=stVG, PG:=stPG);
	PG907:
		fb907(PG:=stVG);
	IG909:
		fb909(IG:=stVG, PG:=stPG);
	PG925:
		fb925(VG:=stVG);
	ELSE
		(* Now, since we don't know what gauge type we're dealing with, we want to make sure to reset all the gauge parameters, otherwise we may be left with stale information *)
	stVG.rPRESS := 760;
	stVG.xAT_VAC := FALSE;
	stVG.xPRESS_OK := FALSE;
	stVG.xHV_SW := FALSE;
		
END_CASE

iq_astGauges[LIMIT(0 ,i_iIndex, gc_iSizeOfGGOArray)] := stVG;
iq_axHV_RO[LIMIT(0,WORD_TO_INT(stVG.wHV_RO),gc_iSizeOfGGOArray)]:=stVG.xHV_DIS;

END_FUNCTION_BLOCK

// POUs/Functions/Gauge FB/FB_GGO_dep
FUNCTION_BLOCK FB_GGO_dep
VAR_IN_OUT
	iq_astGauges: ARRAY[0..50] OF ST_VG;
	iq_axHV_RO: ARRAY[0..50] OF BOOL;
END_VAR
VAR_INPUT
	i_iIndex: INT;
END_VAR
VAR
	rMinPressure_925: REAL := 9E-06;
	rMinPressure_903: REAL := 5E-11;
	rMinPressure_909: REAL := 3E-10;
	rMinPressure_907: REAL := 1E-03;
	rMinPressure_722B: REAL := 0.5;
	
	rV: REAL;
	rA: REAL := 3.29;
	rB: REAL := 24.98;
	rC: REAL := 0.98;
	rV_0: REAL := 0.3752;
	rD: REAL := 4.929;
	rF: REAL := 1.6E-06;
	rG: REAL := -225;
	rH: REAL := 2.0253;
	rK: REAL := 0.52703;
	rFun: REAL;
	xB_FULL_SCALE: BOOL;
	xB_1000_MINVAL: BOOL;
	xB_1_MINVAL: BOOL;
	tonGaugeTurnOnTmr: TON;
	stPG: ST_VG;
	stIG: ST_VG;
	VG: INT;
	H2E_GPI00: INT;
END_VAR

(* This function block is used to calculate the pressure from the analog input voltage and to provide protection and automatic turn on of ion gauges.
 It also manages the turn on fo the AT_VAC boolean, and checks to make sure the pressure is good *)

(* Full-scale pressure conversion factor *)

(* Real-value voltage calculation *)
(* Generic expression for pressure in the MKS systems

P = 10^(V/0.6-12)

722B = 0
903 = 1
907 = 2
909 = 3
925 = 4

*)



(* Check that it is an ion gauge *)
IF iq_astGauges[i_iIndex].iTYPE = 1 OR iq_astGauges[i_iIndex].iTYPE = 3 THEN

	stIG := iq_astGauges[i_iIndex];
	rV := 10*INT_TO_REAL(stIG.iPRESS_R)/32767;
	
	(* Protection Gauge *)
	IF WORD_TO_INT(stIG.wPG) <= g_iSizeOfGGOArray THEN
	(* Check pressure gauge type before assignment *)
	(* Add high pressure gauge types here *)
		IF iq_astGauges[stIG.wPG].iTYPE = 0 OR //722B
		iq_astGauges[stIG.wPG].iTYPE = 2 OR //907
		iq_astGauges[stIG.wPG].iTYPE = 4 THEN //925
			stPG := iq_astGauges[stIG.wPG];
		END_IF
	
	ELSE
		//Default to allow the IG to turn on
		stPG.rPRESS := 1E-3;
		stPG.xPRESS_OK := TRUE;
	END_IF

	(* Protection Functions *)
	(* If the PG pressure is greater than the IG.PRO_SP then the gauge is disabled *)
	(* If the PG pressure is less than the IG.PRO_SP then the gauge is enabled *)
	(* This FB also implements some hysteresis sof the gauge doesn't have rapid power cycling while near the turn on boundary *)


	IF stPG.rPRESS < stIG.rPRO_SP AND stPG.xPRESS_OK THEN
		stIG.xHV_DIS := stIG.xHV_SW;
	ELSIF stIG.xHV_DIS THEN
		IF stIG.rPRESS > stIG.rPRO_SP + stIG.rHYS_PR OR stPG.rPRESS > stIG.rPRO_SP + stIG.rHYS_PR THEN
			stIG.xHV_DIS := FALSE;
			stIG.xHV_SW := FALSE;
		END_IF
	ELSE
		stIG.xHV_DIS := FALSE;
		stIG.xHV_SW := FALSE;
	END_IF

(* Pressure OK check *)
	IF  stIG.iTYPE = 1 THEN
		stIG.rPRESS := LREAL_TO_REAL(EXPT(10, rV-11));
		stIG.xPRESS_OK := ((stIG.rPRESS > rMinPressure_903) AND stIG.xHV_DIS AND stIG.xTurnOnTime) OR stIG.xBAKEOUT;
		tonGaugeTurnOnTmr(IN := stIG.xHV_DIS, PT := T#10s, Q => stIG.xTurnOnTime);

		(* Setpoint evaluation *)
		stIG.xAT_VAC := (stIG.xPRESS_OK AND (stIG.rPRESS < stIG.rVAC_SP)) OR stIG.xBAKEOUT;

(* Pressure OK check *)
	ELSIF stIG.iTYPE = 3 THEN
		stIG.rPRESS := LREAL_TO_REAL(EXPT(10, rV-10));
		stIG.xPRESS_OK := (stIG.rPRESS > rMinPressure_909) AND stIG.xHV_DIS OR stIG.xBAKEOUT;

		(* Setpoint evaluation *)
		stIG.xAT_VAC := stIG.xPRESS_OK AND (stIG.rPRESS < stIG.rVAC_SP) OR stIG.xBAKEOUT;
	END_IF

	(* Copying the calc back over *)
	iq_astGauges[i_iIndex] :=  stIG;

ELSE

 	stPG := iq_astGauges[i_iIndex];
	IF stPG.iTYPE = 0 THEN

		(* Real-value voltage calculation *)
		
		rMinPressure_722B := stPG.rFULL_SCALE * 5E-4;
		

		rV :=MAX((10*INT_TO_REAL(stPG.iPRESS_R)/32767),0);
		stPG.rPRESS := (stPG.rFULL_SCALE/10)*rV;
		
		(* Pressure OK check *)
		stPG.xPRESS_OK := (stPG.rPRESS > rMinPressure_722B);

		(* Setpoint evaluation *)
		stPG.xAT_VAC := stPG.xPRESS_OK AND (stPG.rPRESS < stPG.rVAC_SP);

	ELSIF stPG.iTYPE = 2 THEN

		rV := 10*INT_TO_REAL(stPG.iPRESS_R)/32767;

		IF rV > 0.38 AND rV < 4.85 THEN
			stPG.rPRESS := LREAL_TO_REAL(EXPT((rA/((rB/(EXPT(rV,2)-EXPT(rV_0,2))-1))), 1/rC));
		ELSIF rV > 4.85 AND rV< 5.18 THEN
			stPG.rPRESS := LREAL_TO_REAL(SQRT(((rV-rD)+SQRT(EXPT((rV-rD),2)-4*rF*rG))/(2*rF)));
		ELSIF rV > 5.18 THEN
			stPG.rPRESS := EXP((rV-rH)/rK);
		ELSIF rV <= 0.38 THEN
			stPG.rPRESS := rMinPressure_907;
		END_IF

		(* Protection Functions *)
		(* If the voltage is less than 1mV the gauge is probably not plugged in, or has an issue *)

		(* Pressure OK check *)
		stPG.xPRESS_OK := (rV > 0.01) OR stPG.xBAKEOUT;

		(* Setpoint evaluation *)
		stPG.xAT_VAC := (stPG.xPRESS_OK AND (stPG.rPRESS < stPG.rVAC_SP)) OR stPG.xBAKEOUT;

	ELSIF stPG.iTYPE = 4 THEN

		rV := 10*INT_TO_REAL(stPG.iPRESS_R)/32767;

		IF rV > 1 THEN
			stPG.rPRESS := LREAL_TO_REAL(EXPT(10, rV-6));
		ELSE
			stPG.xPRESS_OK := FALSE;
		END_IF

		(* Protection Functions *)
		(* If the PG pressure is greater than the IG.PRO_SP then the gauge is disabled *)
		(* If the PG pressure is less than the IG.PRO_SP then the gauge is enabled *)
		(* This FB also implements some hysteresis so the gauge doesn't have rapid power cycling while near the turn on boundary *)

		(* Pressure OK check *)
		stPG.xPRESS_OK := (stPG.rPRESS > rMinPressure_925);

		(* Setpoint evaluation *)
		stPG.xAT_VAC := stPG.xPRESS_OK AND (stPG.rPRESS < stPG.rVAC_SP);

ELSE

(* Now, since we don't know what gauge type we're dealing with, we want to make sure to reset all the gauge parameters, otherwise we may be left with stale information *)
	stPG.rPRESS := 760;
	stPG.xAT_VAC := FALSE;
	stPG.xPRESS_OK := FALSE;
	stPG.xHV_SW := FALSE;


END_IF

	(* Copying the calc back over *)
	iq_astGauges[i_iIndex] :=  stPG;

END_IF

//copy the high voltage status over.
iq_axHV_RO[iq_astGauges[i_iIndex].wHV_RO]:=iq_astGauges[i_iIndex].xHV_DIS;

END_FUNCTION_BLOCK

// POUs/Functions/Pumps/FB_EbaraDryPump
FUNCTION_BLOCK FB_EbaraDryPump
VAR_INPUT
	i_stBPGauge	:	ST_VG; //booster pump interlock gauge
	i_xVlvOpn	:	BOOL; //valve(s) to main system load are open
END_VAR
VAR_OUTPUT
END_VAR
VAR_IN_OUT
	stPump	:	ST_EbaraDryPump; //Ebara dry pump structure
END_VAR
VAR
END_VAR

(* Ebara Dry Pump Control Routine
A. Wallace
2016-4-29
Applicable to:
EV-S20
EV-S50
EV-S100
EV-S200

Does basic controls for the pump. Starts booster pump when appropriate. Turns off pump
in the event of errors/ warnings. Provides interlocking interface.

Main Pump Operational Note:
Ebara recommends that the pump be exposed to the full system load after the main pump is running.

Booster Pump Operational Note:
The booster pump can either be started automatically by the pump itself (probably based on a timer?)
or it can be started by the PLC. The pressure setpoint is by default 30T. It may be wise to make
sure the pump was exposed to the full system load before starting the booster.

*)

//Mapping

// These are normally closed inputs
stPump.xErr := NOT stPump.i_xAlarm;
stPump.xWrn := NOT stPump.i_xWarning;


//Interlock and error/warning
stPump.xIlk :=  stPump.xExtIlk AND NOT (stpump.xErr OR stpump.xWrn);

//Start/ Stop the pump
IF stpump.xIlk THEN
	stpump.q_xMPStart := stpump.i_xRunSW;
ELSE
	stpump.q_xMPStart := stpump.i_xRunSW := FALSE;
END_IF

//Booster pump
stpump.xBPIlk := i_xVlvOpn AND stpump.i_xMPStatus AND (i_stBPGauge.rPRESS < stpump.rBPIlkSP) AND i_stbpgauge.xPRESS_OK;
stpump.tonBP(IN:=stpump.xBPIlk);
stpump.q_xBPStart := stpump.tonBP.Q;

END_FUNCTION_BLOCK

// POUs/MAIN
PROGRAM MAIN
VAR
	tpImAPLC : TP;
	stDiag	:	ST_fbDiagnostics;
	valu: INT;
END_VAR

////////////////////////////////////////////////////////////
// Logger test code
tpImAPLC();
IF NOT tpImAPLC.Q THEN
	fbLogMessage(i_sMsg:='Hello world, I am a PLC', i_eSevr:=Info, i_eSubsystem:=E_Subsystem.VACUUM);
	tpImAPLC(IN:= FALSE ); tpImAPLC(IN:= TRUE);
END_IF

////////////////////////////////////////////////////////////
// This gives you an increment at the same time as you get the current index value.
valu := stDiag.resultIdx.ValInc();

END_PROGRAM

// POUs/LOGGER
PROGRAM LOGGER
VAR
	fbLogger	:	FB_Logger;
END_VAR

fbLogger();

END_PROGRAM

// POUs/Logger/FB_Logger
FUNCTION_BLOCK FB_Logger
VAR_INPUT
	i_CloseSocket	:	BOOL := FALSE;
	i_bReset		:	BOOL := FALSE;
END_VAR
VAR
	fbUDPSocketManager	:	FB_ConnectionlessSocket;
	udpSocket			:	T_HSOCKET;
	fbUDPSocketSend		:	FB_SocketUdpSendTo;
	sOutgoingMesg		:	T_MaxString;
	eState				:	E_MessengerState;
	stDiag				:	ST_fbDiagnostics;
	rtReset				:	R_TRIG;
	fbGetSystemTime		:	FB_LocalSystemTime := (bEnable := TRUE);
	fbGetHostName		:	FB_GetHostName := (bExecute := TRUE, sNetID := '');
	ctuSentSomething	:	CTU := (PV := 100);
	rtSocketSendErr		:	R_TRIG;
END_VAR
VAR CONSTANT

END_VAR

(* Syslog Logger
A. Wallace 2016-9-3

This is used to pass PLC notification messeges to a syslog server.

This POU constantly attempts to send out messages from the global buffer.
*)

gfbBuffer.pBuffer := ADR(gMesgBuffer); 
gfbBuffer.cbBuffer:= SIZEOF(gMesgBuffer);

fbGetSystemTime(); 
IF fbGetSystemTime.bValid THEN
	gsCurrentTime := SYSTEM_TIME_TO_RFC3339(fbGetSystemTime.systemTime);
ELSE
	gsCurrentTime := cNILVALUE;
END_IF

fbGetHostName();
IF NOT (fbGetHostName.bBusy OR fbGetHostName.bError) THEN
	gsHostName := fbGetHostName.sHostName;
ELSE
	gsHostName := cNILVALUE;
END_IF

IF i_CloseSocket THEN 
	eState := CloseSocket; 
END_IF

rtReset(CLK:=i_bReset);
IF rtReset.Q THEN
	eState := CreateSocket;
	i_bReset R= i_bReset;
END_IF

rtSocketSendErr(CLK:=fbUDPSocketSend.bError);

CASE eState OF
	Init:
		;
	CreateSocket:
		fbUDPSocketManager.nLocalPort := g_udpSyslog;
		fbUDPSocketManager.bEnable := TRUE;
		
		IF fbUDPSocketManager.eState = eSOCKET_CREATED THEN
			eState := Active;
		ELSIF fbUDPSocketManager.bError THEN
			eState := Err;
			fbUDPSocketManager.bEnable := FALSE;
			stDiag.fString( sOut=>stDiag.asResults[stDiag.resultIdx.ValInc()], sFormat:='Socketmanger error in createsocket: %d', arg1:=F_UDINT(fbUDPSocketManager.nErrID));
		ELSE
			eState := Err;
			stDiag.fString( sOut=>stDiag.asResults[stDiag.resultIdx.ValInc()], sFormat:='Something else happened in createsocket -> error');
		END_IF
	Active:
		IF fbUDPSocketManager.eState = eSOCKET_TRANSIENT  OR 
			fbUDPSocketManager.bError THEN
			eState := Err; 
			stDiag.fString( sOut=>stDiag.asResults[stDiag.resultIdx.ValInc()], sFormat:='Socketmanager error in active: %d', arg1:=F_UDINT(fbUDPSocketManager.nErrId));
		END_IF
		
		// While the socket is active, go ahead and send whatever is in the buffer
		IF rtSocketSendErr.Q THEN
			eState := Err;
			stDiag.fString( sOut=>stDiag.asResults[stDiag.resultIdx.ValInc()], sFormat:='Socket send error: %d', arg1:=F_UDINT(fbUDPSocketSend.nErrId));
		ELSIF gfbBuffer.nCount > 0 AND NOT fbUDPSocketSend.bBusy THEN
			gfbBuffer.A_RemoveHead(getValue=>sOutgoingMesg);
			fbUDPSocketSend.bExecute := TRUE; //reset in the action after busy goes true
			IF sOutgoingMesg <> '' THEN
				ctuSentSomething(CU:=TRUE);
			END_IF
		ELSIF gfbBuffer.nCount = 0 OR fbUDPSocketSend.bBusy THEN
			stDiag.fString( sOut=>stDiag.asResults[stDiag.resultIdx.ValInc()], sFormat:='Waiting to send');
			ctuSentSomething(CU:=FALSE);
		ELSE
			eState := Err;
			stDiag.fString( sOut=>stDiag.asResults[stDiag.resultIdx.ValInc()], sFormat:='Something else happened in active -> error');
		END_IF
		
	CloseSocket:
		fbUDPSocketManager.bEnable R= i_CloseSocket;
		IF fbUDPSocketManager.eState = eSOCKET_CLOSED THEN
			eState := Init;
		ELSIF fbUDPSocketManager.bBusy AND NOT fbUDPSocketManager.bEnable THEN
			;
		ELSIF fbUDPSocketManager.bError THEN
			eState := Err;
		ELSE
			eState := Err;
		END_IF
	Err:
		eState := Init;
		stDiag.asResults[stDiag.resultIdx.ValInc()] := 'Moving back to Init state from Error';
END_CASE



Manager();
SocketSendTo();

ACTION Manager:
fbUDPSocketManager(hSocket => udpSocket);
END_ACTION

ACTION SocketSendTo:
fbUDPSocketSend.hSocket := udpSocket;
fbUDPSocketSend.sRemoteHost := g_psLogHost;
fbUDPSocketSend.nRemotePort := g_udpSyslog;
fbUDPSocketSend.pSrc := ADR(sOutgoingMesg);
fbUDPSocketSend.cbLen := SIZEOF(sOutgoingMesg);
fbUDPSocketSend();
fbUDPSocketSend.bExecute R= fbUDPSocketSend.bBusy;
END_ACTION

END_FUNCTION_BLOCK

// POUs/Logger/SYSTEM_TIME_TO_RFC3339
FUNCTION SYSTEM_TIME_TO_RFC3339 : STRING
VAR_INPUT
	tCurrentTime	:	TIMESTRUCT;
END_VAR
VAR
END_VAR

SYSTEM_TIME_TO_RFC3339 := CONCAT(REPLACE(SYSTEMTIME_TO_STRING(tCurrentTime), 'T', 1, 11), 'Z');

END_FUNCTION

// POUs/Functions/Pumps/FB_PTM_Agilent
FUNCTION_BLOCK FB_PTM_Agilent
VAR_IN_OUT
	iq_stPtm	:	ST_PTM;
END_VAR
VAR_INPUT
END_VAR
VAR_OUTPUT
END_VAR
VAR
	xRunOk	:	BOOL;
END_VAR

(* Basic Agilent Turbo Controls *)
(* A. Wallace, 2015-7-15 *)


(* Interlock Sum *)
xRunOk := iq_stPtm.xExtRunOk AND NOT iq_stPtm.xFault;

(* Mask the at speed bit if fault is true 
done for versions of the interface cable where
at speed gets its power from from the beckhoff term*)
IF iq_stPtm.xFault THEN
	iq_stPtm.i_xAtSpd := FALSE;
END_IF

(* Basic pump supervisory section *)
IF xRunOk THEN
	iq_stPtm.q_RunDO := iq_stPTM.i_xRunSW;
ELSE
	iq_stPtm.i_xRunSW:=FALSE;
	iq_stPtm.q_RunDO:=FALSE;
END_IF

END_FUNCTION_BLOCK

// POUs/Functions/Pumps/FB_PTM_Ebara
FUNCTION_BLOCK FB_PTM_Ebara
VAR_IN_OUT
	iq_stPTM : ST_EbaraPTM;
END_VAR
VAR_INPUT
	i_iADCBits : UINT := 15;
	i_iRawSpeed: INT; //Should come from PLC Soft IO.
END_VAR
VAR_OUTPUT
END_VAR
VAR
	TOF_START: TOF := (PT:=T#0.5S); //Manual states momentary switches need to be closed for >= 0.3s
	TOF_STOP: TOF := (PT:=T#0.5S);
	TOF_RESET: TOF :=(PT:=T#0.5S);
END_VAR

(* Ebara ETC control FB
Scott Stubbs & Alex W.
*)

(* Switch processing *)
TOF_START.IN := iq_stPTM.i_xStart;
TOF_START();
TOF_STOP.IN  := iq_stPTM.i_xStop;
TOF_STOP();
TOF_RESET.IN := iq_stPTM.i_xReset;
TOF_RESET();

//Normally closed fault handling
iq_stPTM.xFault := NOT iq_stPTM.i_xNCFault;

(* Simple protection reset *)
IF iq_stPTM.xExtRunOk THEN
	iq_stPTM.q_xProtection:=TRUE;
END_IF

(* Basic pump supervisory section *)
	(* If override mode, ignore everything else *)
IF iq_stPTM.i_xOverride THEN
	IF TOF_START.Q THEN
	iq_stPTM.q_RunDO:=TRUE;
	ELSIF TOF_STOP.Q THEN
		iq_stPTM.q_RunDO:=FALSE;
	END_IF
	//Handle faults - the way the Ebara cable is done, xFault is normally closed
ELSIF iq_stPTM.xFault OR (iq_stPTM.q_RunDO AND NOT iq_stPTM.xExtRunOk) THEN
	iq_stPTM.q_RunDO:=FALSE;
	iq_stPTM.q_xProtection:=FALSE;
	//And one for when we need to start the pump normally. Only allows pump to be started if ILK ok.
ELSIF TOF_START.Q AND iq_stPTM.xExtRunOk THEN
	iq_stPTM.q_RunDO:=TRUE;
	iq_stPTM.q_xStart:=TOF_START.Q;
//One section for when pump is told to stop
ELSIF TOF_STOP.Q THEN
		iq_stPTM.q_RunDO:=FALSE;
END_IF 

iq_stPTM.q_xReset:=TOF_RESET.Q; //No need for a conditional on these, code below takes care of it
iq_stPTM.q_xStop:=TOF_STOP.Q;
//Reset the start switch after processing
IF iq_stPTM.q_RunDO THEN
	iq_stPTM.q_xStart := TOF_START.Q;
END_IF

(* Pump speed calculation *)
IF iq_stPTM.i_iRawSpeed / (EXPT(2,i_iADCBits)-1) * 10 >= 0.2 THEN //Speed reading appears to zero at ~0.16V
iq_stPTM.i_iCurSpd := LREAL_TO_DINT(iq_stPTM.i_iRawSpeed/(EXPT(2,i_iADCBits)-1)*67000);
//V (AI/(2^{# ADC bits} -1 ) * 10[ADC 10V scaling]) * (33600 [Max RPM] - 100) / 5
ELSE
	iq_stPTM.i_iCurSpd := 0;
END_IF

END_FUNCTION_BLOCK

// POUs/Functions/Pumps/FB_PTM_LeyboldTD20Classic
FUNCTION_BLOCK FB_PTM_LeyboldTD20Classic
VAR_IN_OUT
	iq_stPTM : ST_LeyboldPTM;
END_VAR
VAR_INPUT
END_VAR
VAR_OUTPUT
END_VAR
VAR
	rtReset	:	R_TRIG;
END_VAR

(* Leybold TD20 Classic FB
A. Wallace
NOTE: This FB should be instanced for each pump. It relies on a
persistent state for reseting faults.
*)

//Faults
////////////////////////////
	rtReset(CLK:=iq_stPTM.i_xReset);
	iq_stPTM.xFault R= rtReset.Q;
	iq_stPTM.xFault S= iq_stPTM.i_xTempFault OR NOT iq_stPTM.i_xNCError;

	iq_stPTM.xWarn R= rtReset.Q;
	iq_stPTM.xWarn S= iq_stPTM.xCommTimeout;

(* Basic pump supervisory section *)
IF iq_stPTM.xExtRunOk AND NOT iq_stPTM.xFault THEN
	iq_stPTM.q_RunDO:=iq_stPTM.i_xRunSW;
ELSE
	iq_stPTM.i_xRunSW:=FALSE;
	iq_stPTM.q_RunDO:=FALSE;
END_IF

END_FUNCTION_BLOCK

// POUs/Functions/Pumps/FB_PTM_MagDriveDigital
FUNCTION_BLOCK FB_PTM_MagDriveDigital
VAR_IN_OUT
	iq_stPtm	:	ST_OerlikonPTM;
END_VAR
VAR_INPUT
END_VAR
VAR_OUTPUT
END_VAR
VAR
	xRunOk	:	BOOL;
	tofRemoteDelay	:	TOF;
	
END_VAR

(* Basic MagDrive Digital Turbo Controls *)
(* A. Wallace, 2015-7-15 *)

tofRemoteDelay(IN:=iq_stPtm.q_RunDO, PT:=T#5S);

iq_stPtm.q_xRemote := tofRemoteDelay.Q;

(* Interlock Sum *)
xRunOk := iq_stPtm.xExtRunOk AND NOT iq_stPtm.xFault;

(* Basic pump supervisory section *)
IF xRunOk THEN
	iq_stPtm.q_RunDO := iq_stPTM.i_xRunSW;
ELSE
	iq_stPtm.i_xRunSW:=FALSE;
	iq_stPtm.q_RunDO:=FALSE;
END_IF

END_FUNCTION_BLOCK

// POUs/Functions/Pumps/FB_PTM_Pfeiffer
FUNCTION_BLOCK FB_PTM_Pfeiffer
VAR_IN_OUT
	iq_stPTM : ST_PfeifferPTM;
END_VAR
VAR_INPUT
END_VAR
VAR_OUTPUT
END_VAR
VAR
END_VAR

(* Basic pump supervisory section *)
IF iq_stPTM.xExtRunOk AND NOT (iq_stPTM.xFault OR iq_stPTM.i_xTempFault) THEN
	iq_stPTM.q_RunDO:=iq_stPTM.i_xRunSW;
ELSE
	iq_stPTM.i_xRunSW:=0;
	iq_stPTM.q_RunDO:=FALSE;
END_IF

END_FUNCTION_BLOCK

// POUs/Functions/Valve FB/F_TURBO_VRC_ILK
FUNCTION F_TURBO_VRC_ILK : BOOL
VAR_INPUT

	i_xHiVac 	: BOOL;
	i_xRunPTM	: BOOL;
	i_xFLVac	: BOOL;

END_VAR
VAR

	rHysterisis : REAL := 0;

	xInterlock: BOOL;
	rTolerance: REAL := 20;
END_VAR

(* Close the vic if the roughing pump pirani loses its at-vac setpoint while the turbo is pumping *)
F_TURBO_VRC_ILK := (NOT i_xHiVac AND NOT i_xRunPTM AND NOT i_xFLVac) OR
					(NOT i_xRunPTM AND i_xFLVac) OR
					(i_xRunPTM AND i_xFLVac);

END_FUNCTION

// POUs/Functions/Valve FB/F_VALVE_REL_ILK
FUNCTION F_VALVE_REL_ILK : BOOL
VAR_INPUT
	i_stUSG	:	ST_VG;
	i_stDSG	:	ST_VG;
	//Orders of magnitude allowed between up/downstream pressures for valve to open. Must be real positive integer.
	i_iOrdersMagnitude: INT;
END_VAR
VAR
	rPressRatio : REAL;
	rMaxRatioAllowed	:	LREAL := EXPT(10,i_iOrdersMagnitude);
	rMinRatioAllowed	:	LREAL := EXPT(10,(-i_iOrdersMagnitude));
END_VAR

(* OK, this is going to be a general-use function that will return whether the ratio of the pressures given is less than x orders of magnitude.
True iff 10^(-x) < a/b < 10^x.  Simple, right?  Just make sure it gets a positive order of magnitude and the pressures aren't 0. ~Scott *)   

(* Find ratio *)

IF i_stDSG.rPRESS <> 0 THEN
	rPressRatio := i_stUSG.rPRESS / i_stDSG.rPRESS;

	F_VALVE_REL_ILK := rPressRatio < rMaxRatioAllowed AND rMinRatioAllowed < rPressRatio;
ELSE
	F_VALVE_REL_ILK := FALSE;
END_IF

END_FUNCTION

// POUs/Functions/Valve FB/F_VRC_DIODE_ILK
FUNCTION F_VRC_DIODE_ILK : BOOL
VAR_INPUT

	i_stPGA : ST_VG;
	i_stPGB	: ST_VG;

END_VAR
VAR

	rHysterisis : REAL := 0;

	xInterlock: BOOL;
	rTolerance: REAL := 20;
END_VAR

(* The principle is simple, a VRC should never open when B side pressure is greater than the A side pressure. *)
rTolerance := 20;
F_VRC_DIODE_ILK := ((i_stPGA.rPRESS + rTolerance >= i_stPGB.rPRESS + rHysterisis) OR i_stPGA.xBAKEOUT) AND i_stPGA.xPRESS_OK AND i_stPGB.xPRESS_OK;

(* OK it gets a bit more complicated with hysterisis,

Now, if the F_VIC_DIODE_ILK is FALSE then some hysterisis is added to the B side. But if it's OK then we just stick with making sure that the A side is greater than the B side

*)
(*
IF NOT F_VIC_DIODE_ILK THEN
Hysterisis := 40;
ELSE
Hysterisis := 0;
END_IF
*)

END_FUNCTION

// POUs/Functions/Valve FB/FB_VCC
FUNCTION_BLOCK FB_VCC
VAR_IN_OUT

	iq_stValve : ST_VCC;

END_VAR
VAR_INPUT

END_VAR
VAR_OUTPUT
END_VAR
VAR

tonOvrd	:	TON;
tonDelOK : TON;
rtOK	:	R_TRIG;

END_VAR


IF NOT iq_stValve.xOPN_OK THEN
iq_stValve.xOPN_SW := FALSE;
END_IF

(* Override logic *)
(* Goal: give ability to override, but do so in a way that people won't forget it.
Solution: Override only after ten seconds of override, protect against blips,
when the valve permission goes true for more than ten seconds consistently, remove override
*)

tonDelOK(IN:=iq_stValve.xOPN_OK, PT:=T#10S);
rtOK(CLK:=tonDelOK.Q);
IF rtOK.Q THEN iq_stValve.xOvrdOpn :=FALSE; END_IF

//Override timer
tonOvrd(IN:=iq_stValve.xOvrdOpn, PT:=T#10S);

(* Here's where the valve opens *)
iq_stValve.xOPN_DO := (iq_stValve.xOPN_SW AND iq_stValve.xOPN_OK) OR (tonOvrd.Q AND g_stSystem.xOverrideMode);

END_FUNCTION_BLOCK

// POUs/Functions/Valve FB/FB_VCN
FUNCTION_BLOCK FB_VCN
VAR_INPUT
	i_xExtIlk	:	BOOL; //External Interlock
	i_ReqPos	:	BOOL; //Requested position
END_VAR
VAR_OUTPUT
END_VAR
VAR_IN_OUT
	iq_stVCN	:	ST_VCN; //Needle valve structure
END_VAR
VAR
	// Requested voltage
	rReqVoltage: REAL := 0;
END_VAR
VAR CONSTANT
	rOpenVoltage	:	REAL := 9.1; // From the EVR 116 manual
	rCloseVoltage	:	REAL := 0.4;
END_VAR

(* Needle valve control FB
A. Wallace 2016-7-21

This FB should be used as a low level control block.

It provides:

Valve position ceiling
Interlock
Scaling

It is not intended for:
Closed-loop control

It could be used for:
Valve position/flow linearization

Note: Raw position calc is based on 0.5 to 9V span, 32767 bits
*)




// Interlocking
iq_stVCN.xIlk := i_xExtIlk;

IF iq_stVCN.xIlk THEN
	
	IF iq_stVCN.eValveControl = OpenValve THEN
		iq_stVCN.rReqPosition := iq_stVCN.rUpperLimit;
	ELSIF iq_stVCN.eValveControl = CloseValve THEN
		iq_stVCN.rReqPosition := 0;
	ELSE
		 ;
	END_IF

	//Raw position calc
	iq_stVCN.rReqPosition := LIMIT(0, iq_stVCN.rReqPosition, iq_stVCN.rUpperLimit);
	rReqVoltage := iq_stVCN.rReqPosition * (rOpenVoltage-rCloseVoltage)/100 + rCloseVoltage;
	rReqVoltage := LIMIT(rCloseVoltage, rReqVoltage, rOpenVoltage); //The requested voltage should remain within this range
	iq_stvcn.q_iRawPosition := REAL_TO_INT( 32767/10 * rReqVoltage);	
ELSE
	iq_stvcn.q_iRawPosition := 0;
	iq_stVCN.rReqPosition := 0;
	iq_stVCN.eValveControl := CloseValve;
END_IF

END_FUNCTION_BLOCK

// POUs/Functions/Valve FB/FB_VGC
FUNCTION_BLOCK FB_VGC
VAR_IN_OUT

	iq_stValve : ST_VGC;

END_VAR
VAR_INPUT

	i_stUSG	:	ST_VG;
	i_stDSG	:	ST_VG;

	i_xDis_DPIlk : BOOL := FALSE;	// Obsolete
	rDiffPressAllowed	:	REAL := 22.5; // Torr, Default value comes from Vat Valve Manual
END_VAR
VAR_OUTPUT
END_VAR
VAR

	rDiffPress : REAL;

	  

	VGC_State : E_VGC;

	xFirstPass	:	BOOL;
	fbFSInit		:	R_TRIG;
	
	tonDelOK : TON;
	rtOK	:	R_TRIG;
	tonOvrd	:	TON;
	
	tDelOK	:	TIME := T#10S;
	tOvrd	:	TIME := T#10s;
END_VAR

(* Vacuum gate valve
A. Wallace
16-10-29

A gate valve isolates vacuum volumes. Ideally it can be opened when a system is vented
to allow for faster pumping, and will close when high vacuum is lost.

The following behavior is good for valves in something like a gas attenuator.
This function block does the following:
1. The valve can be opened when the difference between the pressures on both sides is
less than the maximum differential pressure.
2. This rule persists until the pressures on both sides are lower than the vacuum-setpoint.
3. Once at-vac, the valve will close if the pressure on either side rises above the setpoint.

Alternatively, the differential pressure interlock can be disabled so the valve may only be opened
if the pressure on both sides is lower than the at-vacuum-setpoint. You want this behavior if 
the valve is to be used in a UHV section.

Hysteresis is employed to ensure a smooth transition from vented/pumping down, to at-vac.

Finally, an override system is built in so you can bypass all the interlocking logic and 
get back online.
*)


fbFSInit( CLK := TRUE,
			Q => xFirstPass);

(* On first PLC pass, put valve into vented state, which implies a closed valve *)
IF xFirstPass THEN
VGC_State := Vented;
iq_stValve.xOPN_SW := FALSE;
END_IF

// Update hysteresis
///////////////////////////////////////////////////
IF iq_stValve.rAT_VAC_SP_LAST <> iq_stValve.rAT_VAC_SP THEN
	iq_stValve.rAT_VAC_SP_LAST := iq_stValve.rAT_VAC_SP;
	iq_stValve.rAT_VAC_HYS := iq_stValve.rHYST_PERC * iq_stValve.rAT_VAC_SP;
END_IF

iq_stValve.rAT_VAC_HYS := LIMIT(0, iq_stValve.rAT_VAC_HYS, iq_stValve.rAT_VAC_SP);
IF iq_stValve.rHYST_PERC <> (iq_stValve.rAT_VAC_HYS / iq_stValve.rAT_VAC_SP) THEN
	iq_stValve.rHYST_PERC := LIMIT(0, (iq_stValve.rAT_VAC_HYS / iq_stValve.rAT_VAC_SP) ,1);
END_IF

// Valve at vacuum check
///////////////////////////////////////////////////
	iq_stValve.xAT_VAC S= i_stUSG.rPRESS < iq_stValve.rAT_VAC_HYS AND i_stDSG.rPRESS < iq_stValve.rAT_VAC_HYS AND i_stUSG.xPRESS_OK AND i_stDSG.xPRESS_OK;
	iq_stValve.xAT_VAC R= i_stUSG.rPRESS < iq_stValve.rAT_VAC_SP AND i_stDSG.rPRESS < iq_stValve.rAT_VAC_SP AND i_stUSG.xPRESS_OK AND i_stDSG.xPRESS_OK;

// Differential pressure check
///////////////////////////////////////////////////
	(* Calc the differential pressure across the valve *)
	rDiffPress := ABS(i_stUSG.rPRESS - i_stDSG.rPRESS);
	
	(* As long as the differential pressure is less than 30mbar, the valve is allowed to open *)
	IF rDiffPress <= rDiffPressAllowed AND i_stUSG.xPRESS_OK AND i_stDSG.xPRESS_OK THEN
		iq_stValve.xDP_OK := TRUE;
	ELSE
		iq_stValve.xDP_OK	:= FALSE;
		(* If the differential pressure is exceeded, even when the valve is open,
		the state is unexpected and triggers a fault, because it suggests that something
		is wrong with the valve, or gauges or mapping or there is a major leak on one side.*)
		VGC_State := ERR_DiffPress;
	END_IF

// Valve state
///////////////////////////////////////////////////
CASE VGC_State OF
	Vented: (* The Vented state is used during pump down *)
		(* Assuming the pump down went well, we are now at vacuum on both sides,
		so we move to the vacuum state, otherwise remain in the vented state *)
		IF iq_stValve.xAT_VAC THEN
		VGC_State := AtVacuum;
		ELSE
		VGC_State := Vented;
		END_IF
	
	AtVacuum:
		IF iq_stValve.xAT_VAC THEN
		(* If both pressure setpoints are made,
		then enable the differential pressure interlock, regardless of the valve state
		assuming we're using some kind of ion gauge where a pressure setpoint cannot be higher than 1E-4 T *)
		VGC_State := AtVacuum;
		ELSE
		
			(* If the valve is open (or in an unknown state) and either gauge is not at it's vacuum setpoint,
			we have a loss of vacuum error *)
			IF (iq_stValve.i_xOpnLS OR (NOT iq_stValve.i_xOpnLS AND NOT iq_stValve.i_xClsLS)) THEN
			VGC_State := ERR_LostVac;
		
			(* Alternatively, if the valve is already closed and we lose pressure on one side,
			it was probably intentional venting, so we calmly move back to venting mode, and
			disable the differential pressure interlock *)
			ELSIF iq_stValve.i_xClsLS THEN
			VGC_State := Vented;
			END_IF
		
		END_IF
	
	ERR_DiffPress:
		VGC_State := Vented;
		iq_stValve.xERR_DifPres := TRUE;
	
	ERR_LostVac:
		VGC_State := Vented;
		iq_stValve.xERR_LstVac := TRUE;
	
	END_CASE




// Interlock evaluation
///////////////////////////////////////////////
iq_stValve.xOPN_OK := iq_stValve.xEXT_OK AND iq_stValve.xAT_VAC;


(* Valve operation *)

(* Reset the EPICS command to open the valve if the interlock is lost *)
IF NOT iq_stValve.xOPN_OK THEN
iq_stValve.xOPN_SW := FALSE;
END_IF

(* Override logic *)
(* Goal: give ability to override, but do so in a way that people won't forget it.
Solution: Override only after ten seconds of override, protect against blips,
when the valve permission goes true for more than ten seconds consistently, remove override
*)

tonDelOK(IN:=iq_stValve.xOPN_OK, PT:=tDelOK);
rtOK(CLK:=tonDelOK.Q);
IF rtOK.Q AND iq_stValve.xOvrdOpn THEN 
iq_stValve.xOvrdOpn :=FALSE;
iq_stValve.xOPN_SW := TRUE; //for seamless transition
END_IF

//Override timer
tonOvrd(IN:=iq_stValve.xOvrdOpn, PT:=tOvrd);

(* Here's where the valve opens *)
iq_stValve.xOPN_DO := (iq_stValve.xOPN_SW AND iq_stValve.xOPN_OK) OR (tonOvrd.Q AND g_stSystem.xOverrideMode);

// Alarm reset
//////////////////////////////////////
ACT_ResetAlarms();

ACTION ACT_ResetAlarms:
iq_stValve.xERR_DifPres R= iq_stValve.xAlmRst;
iq_stValve.xERR_LstVac R= iq_stValve.xAlmRst;
END_ACTION

END_FUNCTION_BLOCK

// POUs/Functions/Valve FB/FB_VGC_NO
FUNCTION_BLOCK FB_VGC_NO
VAR_IN_OUT

	iq_stValve : ST_VGC_NO;

END_VAR
VAR_INPUT

	i_stUSG	:	ST_VG;
	i_stDSG	:	ST_VG;

	i_xDis_DPIlk : BOOL := FALSE; (*Set to true when calling the function to disable the differential pressure interlock *)
	i_rDiffPressAllowed	:	REAL := 22.5;
END_VAR
VAR_OUTPUT
END_VAR
VAR

	rDiffPress : REAL;

	

	VGC_State : E_VGC;

	xFirstPass	:	BOOL;
	fbFSInit		:	R_TRIG;
	
	tonDelOK : TON;
	rtOK	:	R_TRIG;
	tonOvrd	:	TON;

END_VAR

(* Normally Open Gate Valve
This kind of gate valve can usually be found in systems with some kind of delicate window valve, not intended to hold
a full atmosphere.
*)

fbFSInit( CLK := TRUE,
			Q => xFirstPass);

(* On first PLC pass, put valve into vented state, which implies an open valve *)
IF xFirstPass THEN
VGC_State := Vented;
iq_stValve.xCLS_SW := FALSE;
END_IF


(* Calc the differential pressure across the valve *)
rDiffPress := ABS(i_stUSG.rPRESS - i_stDSG.rPRESS);


(* Here's where the Dis_DPIlk can enable or disable the DP interlock code above,
By default the Dis_DPIlk is FALSE, so the valve is interlocked by the external interlocks
and the differential pressure across the valve. *)

IF i_xDis_DPIlk THEN
iq_stValve.xCLS_OK := iq_stValve.xEXT_OK;
ELSE

CASE VGC_State OF

Vented: (* The Vented state is used during pump down *)

(* As long as the differential pressure is less than 30mbar, the valve is allowed to close/ remain closed *)
IF rDiffPress <= i_rDiffPressAllowed AND i_stUSG.xPRESS_OK AND i_stDSG.xPRESS_OK THEN
iq_stValve.xDP_OK := TRUE;
ELSE
iq_stValve.xDP_OK	:= FALSE;
(* If the differential pressure is exceeded, even when the valve is open,
the state is unexpected and triggers a fault, because it suggests that something
is wrong with the valve, or gauges or mapping or there is a major leak on one side.*)
VGC_State := ERR_DiffPress;
END_IF

(* Assuming the pump down went well, we are now at vacuum on both sides,
so we move to the vacuum state, otherwise remain in the vented state *)
IF i_stUSG.xAT_VAC AND i_stDSG.xAT_VAC AND i_stUSG.xPRESS_OK AND i_stDSG.xPRESS_OK THEN
VGC_State := AtVacuum;
ELSE
VGC_State := Vented;
END_IF

AtVacuum:
(* Note for normally open valves, the condition for remaining closed is that the differential pressure
does not exceed some certain value, which comes from the pressure that the window can hold.
*)
IF rDiffPress <= i_rDiffPressAllowed AND i_stUSG.xPRESS_OK AND i_stDSG.xPRESS_OK THEN
(* If both pressure setpoints are made,
then enable the differential pressure interlock, regardless of the valve state
assuming we're using some kind of ion gauge where a pressure setpoint cannot be higher than 1E-4 T *)
iq_stValve.xDP_OK := TRUE;
VGC_State := AtVacuum;
ELSE

	(* If the valve is closed (or in an unknown state) and either gauge is not at it's vacuum setpoint,
	we have a loss of vacuum error *)
	IF (iq_stValve.i_xClsLS OR (NOT iq_stValve.i_xOpnLS AND NOT iq_stValve.i_xClsLS)) AND 
	(NOT i_stUSG.xAT_VAC OR NOT i_stDSG.xAT_VAC) THEN
		VGC_State := ERR_LostVac;
		iq_stValve.xDP_OK := FALSE;

	(* Alternatively, if the valve is already open and we lose vacuum or differential pressure,
	it was probably intentional venting, so we calmly move back to venting mode, and
	disable the differential pressure interlock *)
	ELSIF iq_stValve.i_xOpnLS AND(NOT i_stUSG.xAT_VAC OR NOT i_stDSG.xAT_VAC) THEN
		iq_stValve.xDP_OK := FALSE;
		VGC_State := Vented;
	END_IF

END_IF

ERR_DiffPress:
iq_stValve.xDP_OK := FALSE;
VGC_State := Vented;
iq_stValve.xERR_DifPres := TRUE;

ERR_LostVac:
iq_stValve.xDP_OK := FALSE;
VGC_State := Vented;
iq_stValve.xERR_LstVac := TRUE;

END_CASE

(* In the default state the Valve.CLS_OK depends on both the external and differential pressure interlocks *)
iq_stValve.xCLS_OK := iq_stValve.xEXT_OK AND iq_stValve.xDP_OK;
END_IF

(* Valve operation *)

(* Reset the PLC/EPICS command to open the valve if the interlock is lost *)
IF NOT iq_stValve.xCLS_OK THEN
iq_stValve.xCLS_SW := FALSE;
END_IF

(* Override logic *)
(* Goal: give ability to override, but do so in a way that people won't forget it.
Solution: Override only after ten seconds of override, protect against blips,
when the valve permission goes true for more than ten seconds consistently, remove override
*)

tonDelOK(IN:=iq_stValve.xCLS_OK, PT:=T#10S);
rtOK(CLK:=tonDelOK.Q);
IF rtOK.Q AND iq_stValve.xOvrdCls THEN 
iq_stValve.xOvrdCls :=FALSE;
iq_stValve.xCLS_SW := TRUE;
END_IF

//Override timer
tonOvrd(IN:=iq_stValve.xOvrdCls, PT:=T#10S);

(* Here's where the valve is closed *)
iq_stValve.xCLS_DO := (iq_stValve.xCLS_SW AND iq_stValve.xCLS_OK) OR (tonOvrd.Q AND g_stSystem.xOverrideMode);

ACTION ACT_ResetAlarms:
iq_stValve.xERR_DifPres R= iq_stValve.xAlmRst;
iq_stValve.xERR_LstVac R= iq_stValve.xAlmRst;
END_ACTION

END_FUNCTION_BLOCK

// POUs/Functions/Valve FB/FB_VRC
FUNCTION_BLOCK FB_VRC
VAR_IN_OUT

	iq_stValve : ST_VRC;

END_VAR
VAR_INPUT

END_VAR
VAR_OUTPUT
END_VAR
VAR

tonOvrd	:	TON;
tonDelOK : TON;
rtOK	:	R_TRIG;

END_VAR


IF NOT iq_stValve.xOPN_OK and NOT tonOvrd.Q THEN
iq_stValve.xOPN_SW := FALSE;
END_IF

(* Override logic *)
(* Goal: give ability to override, but do so in a way that people won't forget it.
Solution: Override only after ten seconds of override, protect against blips,
when the valve permission goes true for more than ten seconds consistently, remove override
*)

tonDelOK(IN:=iq_stValve.xOPN_OK, PT:=T#10S);
rtOK(CLK:=tonDelOK.Q);
IF rtOK.Q THEN iq_stValve.xOvrdOpn :=FALSE; END_IF

//Override timer
tonOvrd(IN:=iq_stValve.xOvrdOpn, PT:=T#10S);

(* Here's where the valve opens *)
iq_stValve.xOPN_DO := (iq_stValve.xOPN_SW AND iq_stValve.xOPN_OK) OR (tonOvrd.Q AND g_stSystem.xOverrideMode);

END_FUNCTION_BLOCK

// POUs/Functions/Valve FB/FB_VRC_OK_CLS
FUNCTION_BLOCK FB_VRC_OK_CLS
VAR_IN_OUT

	iq_stValve : ST_VRC;

END_VAR
VAR_INPUT

END_VAR
VAR_OUTPUT
END_VAR
VAR

tonOvrd	:	TON;
tonDelOK : TON;
rtOK	:	R_TRIG;

END_VAR

(* This fumction block is different from the regular VRC in that CLOSING must be permitted. *)
(* Implemented for the funky valve 04 on LAMP *)
IF NOT iq_stValve.xOPN_OK and NOT tonOvrd.Q THEN
iq_stValve.xOPN_SW := FALSE;
END_IF

(* Override logic *)
(* Goal: give ability to override, but do so in a way that people won't forget it.
Solution: Override only after ten seconds of override, protect against blips,
when the valve permission goes true for more than ten seconds consistently, remove override
*)

tonDelOK(IN:=iq_stValve.xOPN_OK, PT:=T#10S);
rtOK(CLK:=tonDelOK.Q);
IF rtOK.Q THEN iq_stValve.xOvrdOpn :=FALSE; END_IF

//Override timer
tonOvrd(IN:=iq_stValve.xOvrdOpn, PT:=T#10S);

(* Here's where the valve opens *)
iq_stValve.xOPN_DO := NOT iq_stValve.xCLS_OK OR ((iq_stValve.xOPN_SW AND iq_stValve.xOPN_OK) OR (tonOvrd.Q AND g_stSystem.xOverrideMode));

END_FUNCTION_BLOCK

// POUs/Functions/FB_EcatDiag
FUNCTION_BLOCK FB_EcatDiag
VAR_INPUT
	///Connect this to an AMSNETID structure as a PLC input. Then link the input to the AMSNETID name in the master info.
	i_AMSNetId: AMSNETID; 
	i_xFirstPass: BOOL;
END_VAR
VAR_OUTPUT
	q_xAllStatesGood: BOOL;
END_VAR
VAR
	sNetId: T_AmsNetId;
	astTermStates: ARRAY[1..256] OF ST_EcSlaveState;
	fbGetAllSlaveStates: FB_EcGetAllSlaveStates;
	ftReset: F_TRIG;
	iterator: INT;
END_VAR

(* 
Ecat bus diagnostic tool
2015-11-4 Alex Wallace
This function block checks the states of all slaves on the ecat bus network, 
it could be modified to export the states of the slaves on an individual basis,
but for now it sets the output boolean true if all slaves are OP and false otherwise.
To start the block provide a falling edge on the first pass boolean input.
*)

//Create the net ID string
sNetID := F_CreateAmsNetId(i_AMSNetId);

//Query the state of all terminals, collect in astTermStates
ftReset(CLK:=fbGetAllSlaveStates.bBusy OR i_xFirstPass);
fbGetAllSlaveStates.bExecute := ftReset.Q;
fbGetAllSlaveStates(sNetId:=sNetId, pStateBuf := ADR(astTermStates), cbBufLen:=SIZEOF(astTermStates));
//Keep checking...

//Cycle through each entry in the array and check if we have anyone not in OP and that the link state is good.
// If so, then set our global IO bad boolean.
IF fbGetAllSlaveStates.nSlaves > 0 THEN
	q_xAllStatesGood := TRUE;
FOR iterator := 1 TO (UINT_TO_INT(fbGetAllSlaveStates.nSlaves) -1) BY 1
	DO
	IF NOT( (astTermStates[iterator].deviceState = EC_DEVICE_STATE_OP) AND (astTermStates[iterator].linkState = EC_LINK_STATE_OK)) THEN
		q_xAllStatesGood := FALSE;
	END_IF
END_FOR
END_IF

END_FUNCTION_BLOCK

// POUs/Functions/FB_Index
FUNCTION_BLOCK FB_Index
VAR_INPUT
	InitVal : INT := 0;
	IncVal : INT := 1;
	UpperLimit	:	INT := 1;
END_VAR
VAR_OUTPUT
	
END_VAR
VAR
	Val	:	INT := InitVal;
END_VAR

(* Index FB
A. Wallace 2016-9-3

Why doesn't beckhoff have this as a builtin type?
*)

;

ACTION Dec:
Val := LIMIT(InitVal, Val - IncVal, UpperLimit);
END_ACTION

ACTION Inc:
// Dont use this, use ValInc
Val := Val + IncVal;
IF Val >  UpperLimit THEN Val := InitVal; END_IF
END_ACTION

METHOD PUBLIC ValInc : INT
VAR_INPUT
END_VAR
ValInc := THIS^.Val;
THIS^.Inc();
END_METHOD

END_FUNCTION_BLOCK

// POUs/Logger/FB_LogMessage
FUNCTION_BLOCK FB_LogMessage
VAR_INPUT	
	i_sMsg	:	STRING;
	i_eSevr	:	E_MesgSevr;
	i_eSubsystem	:	E_Subsystem; //In-lieu of App-name in the RFC-5424
END_VAR
VAR
	i_sPID	:	STRING := cNILVALUE;	//Not currently used
	i_sMSGID	:	STRING := cNILVALUE; //Not currently used
	i_sSD	:	STRING := cNILVALUE; //Not currently used
	fbFormatString		:	FB_FormatString;
	sPRIVAL				: 	T_MaxString := cNILVALUE;
	sPID				: 	T_MaxString := cNILVALUE;
	sSubsystem			: 	T_MaxString := cNILVALUE;
	wSyslogVer			: 	WORD := cwSyslogVer;
	sSD					: 	T_MaxString := cNILVALUE;
	sMsg				: 	T_MaxString := cNILVALUE;
END_VAR

gfbBuffer.putValue := '';
gfbBuffer.pBuffer := ADR(gMesgBuffer);
gfbBuffer.cbBuffer := SIZEOF(gMesgBuffer);

fbFormatString.sFormat := '<%s> %d %s %s %s %s BOM%s';

sPRIVAL := LEFT( WORD_TO_STRING(cwFacility * 8 + i_eSevr), 5);
sPID := cNILVALUE;
sSubsystem := acsSubsystems[i_eSubsystem];
wSyslogVer := cwSyslogVer;
sSD := i_sSD;
sMsg := i_sMsg;
//bad language ahead, sorry
fbFormatString.arg1 := F_STRING(sPRIVAL);
fbFormatString.arg2 := F_WORD(wSyslogVer);
fbFormatString.arg3 := F_STRING(gsCurrentTime);
fbFormatString.arg4 := F_STRING(sSubsystem);
fbFormatString.arg5 := F_STRING(sPID);
fbFormatString.arg6 := F_STRING(sSD);
fbFormatString.arg7 := F_STRING(sMsg);
fbFormatString( sOut=>gfbBuffer.putValue);
gfbBuffer.A_AddTail();

END_FUNCTION_BLOCK
